{attribute 'GeneratedUsingTerminal: EK1960-0000-0021'}
{attribute addProperty BoxType "EK1960-0000-0021"}
{attribute addProperty Id "FSoE_InputsFSoE_Inputs_6CB74C4A47FSoE_OutputsFSoE_Outputs_D808233951"}
{attribute addProperty CRC "69971923"}
{attribute addProperty Size "98"}
TYPE Module_1_FSoE_042BAFD3 :
STRUCT
	{attribute addProperty Name "FSoE_Inputs"}
	FSoE_Inputs  : FSoE_Inputs_6CB74C4A;
	{attribute addProperty Name "FSoE_Outputs"}
	FSoE_Outputs  : FSoE_Outputs_D8082339;
END_STRUCT
END_TYPE

(* stored: Version 1.2.0.0, ProductVersion 3.1.4024.9
   DUT Module_1_FSoE_042BAFD3: Id {05961aa1-aee0-4854-851c-5163cf8c1b9e} *)
